// TIA Portal V18 program export: 1 tag tables, 0 data types, 2 data blocks, 1 code blocks (in call order from the OBs), 0 instance data blocks

VAR_GLOBAL   // PLC tag table "Default tag table"
   System_Byte AT %MB1 : Byte;
   FirstScan AT %M1.0 : Bool;
   DiagStatusUpdate AT %M1.1 : Bool;
   AlwaysTRUE AT %M1.2 : Bool;
   AlwaysFALSE AT %M1.3 : Bool;
   Clock_Byte AT %MB0 : Byte;
   Clock_10Hz AT %M0.0 : Bool;
   Clock_5Hz AT %M0.1 : Bool;
   "Clock_2.5Hz" AT %M0.2 : Bool;
   Clock_2Hz AT %M0.3 : Bool;
   "Clock_1.25Hz" AT %M0.4 : Bool;
   Clock_1Hz AT %M0.5 : Bool;
   "Clock_0.625Hz" AT %M0.6 : Bool;
   "Clock_0.5Hz" AT %M0.7 : Bool;
   MB_Write_Req AT %M10.0 : Bool;
   MB_Read_Req AT %M10.1 : Bool;
   MB_Write_Done AT %M10.2 : Bool;
   MB_Write_Busy AT %M10.3 : Bool;
   MB_Write_Error AT %M10.4 : Bool;
   MB_Read_Done AT %M10.5 : Bool;
   MB_Read_Busy AT %M10.6 : Bool;
   MB_Read_Error AT %M10.7 : Bool;
   MB_Write_Status AT %MW12 : Word;
   MB_Read_Status AT %MW14 : Word;
END_VAR

DATA_BLOCK "DB_MB_Client_Conn"   // DB11
TITLE = DB_MB_Client_Conn
{ S7_Optimized_Access := 'FALSE' }
VERSION : 0.1
// DB communication via Modbus TCP
// stored: AutoNumber false, IsOnlyStoredInLoadMemory false, IsWriteProtectedInAS false
   VAR
      MB_TCP : TCON_IP_v4;
   END_VAR
BEGIN
END_DATA_BLOCK

DATA_BLOCK "DB_MB_Client_Data"   // DB10
TITLE = DB_MB_Client_Data
{ S7_Optimized_Access := 'FALSE' }
VERSION : 0.1
// DB communication via Modbus TCP
// stored: AutoNumber false, IsOnlyStoredInLoadMemory false, IsWriteProtectedInAS false
   VAR
      Send_Words : Array[0..2] of Int;
      Recv_Words : Array[0..9] of Int;
   END_VAR
BEGIN
END_DATA_BLOCK

ORGANIZATION_BLOCK "Main"   // OB1, LAD, ProgramCycle
TITLE = "Main Program Sweep (Cycle)"
{ S7_Optimized_Access := 'TRUE' }
VERSION : 0.1
// stored: AutoNumber true, IsIECCheckEnabled false, SetENOAutomatically false
   VAR_INPUT
      Initial_Call : Bool;   // Initial call of this OB
      Remanence : Bool;   // =True, if remanent data are available
   END_VAR
BEGIN

REGION Network 1
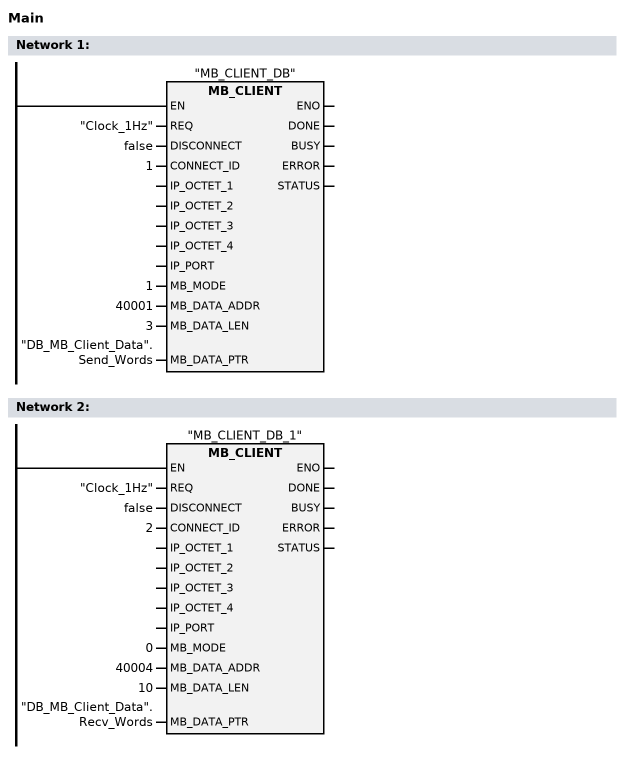
   RUNG wire#powerrail
      { S7_Templates := "[card1200 := 1, card1500 := 0]" } "MB_CLIENT_DB".MB_CLIENT(REQ := "Clock_1Hz", DISCONNECT := false, CONNECT_ID := 1, IP_OCTET_1 :=, IP_OCTET_2 :=, IP_OCTET_3 :=, IP_OCTET_4 :=, IP_PORT :=, MB_MODE := 1, MB_DATA_ADDR := 40001, MB_DATA_LEN := 3, MB_DATA_PTR := "DB_MB_Client_Data".Send_Words, DONE =>, BUSY =>, ERROR =>, STATUS =>)
   END_RUNG
   // the same network as SCL:
   "MB_CLIENT_DB"(REQ := "Clock_1Hz",   // MB_CLIENT
                  DISCONNECT := false,
                  CONNECT_ID := 1,
                  MB_MODE := 1,
                  MB_DATA_ADDR := 40001,
                  MB_DATA_LEN := 3,
                  MB_DATA_PTR := "DB_MB_Client_Data".Send_Words);
END_REGION

REGION Network 2
   RUNG wire#powerrail
      { S7_Templates := "[card1200 := 1, card1500 := 0]" } "MB_CLIENT_DB_1".MB_CLIENT(REQ := "Clock_1Hz", DISCONNECT := false, CONNECT_ID := 2, IP_OCTET_1 :=, IP_OCTET_2 :=, IP_OCTET_3 :=, IP_OCTET_4 :=, IP_PORT :=, MB_MODE := 0, MB_DATA_ADDR := 40004, MB_DATA_LEN := 10, MB_DATA_PTR := "DB_MB_Client_Data".Recv_Words, DONE =>, BUSY =>, ERROR =>, STATUS =>)
   END_RUNG
   // the same network as SCL:
   "MB_CLIENT_DB_1"(REQ := "Clock_1Hz",   // MB_CLIENT
                    DISCONNECT := false,
                    CONNECT_ID := 2,
                    MB_MODE := 0,
                    MB_DATA_ADDR := 40004,
                    MB_DATA_LEN := 10,
                    MB_DATA_PTR := "DB_MB_Client_Data".Recv_Words);
END_REGION
END_ORGANIZATION_BLOCK
